FUNCTION_BLOCK SampleSequence IMPLEMENTS I_Cyclic
VAR
	ThisMover : I_XtsMover;
	LeaveTest: BOOL;
	ArriveTest: BOOL;
	TestMove: BOOL;
	Position: MC_LREAL;
	Velocity: MC_LREAL;
END_VAR

METHOD PUBLIC  Cycle : HRESULT
VAR_INPUT
END_VAR
IF LeaveTest THEN
	ThisMover.TriggerMoverLeave();
END_IF

IF ArriveTest THEN
	ThisMover.TriggerMoverArrive();
END_IF

IF TestMove THEN
	ThisMover.MoveTo(RequiredPosition := Position, MoveVelocity := Velocity, NonModuloMove := FALSE);
	TestMove := FALSE;
END_IF
END_METHOD

PROPERTY MyMover : I_XtsMover
GET
MyMover := ThisMover;
END_GET
SET
ThisMover := MyMover;
END_SET
END_PROPERTY

END_FUNCTION_BLOCK

(* stored: Version 1.1.0.1, ProductVersion 3.1.4026.12
   POU SampleSequence: Id {aeca387d-57da-4277-9b3c-59b22eeb58f8}, SpecialFunc None
   Method Cycle: Id {e67454eb-585e-4a43-aa27-1301f6d081d1}
   Property MyMover: Id {c23dd5f6-58df-442d-9989-7b1384c2b3ac}
   Get Get: Id {b9d1641a-aa56-4f84-90c7-004f2597e2ee}
   Set Set: Id {5ca29307-712f-4ddb-a5e2-33d69141bb16} *)
